{attribute 'GeneratedUsingTerminal: EL3041-0000-0017'}
{attribute addProperty BoxType "EL3041-0000-0017"}
{attribute addProperty Id "AI_StandardAT %I*AI_Standard_Channel_4A3944819WcStateAT %I*WcState_9091E0EB2InfoDataAT %I*InfoData_94A18F5E2"}
{attribute addProperty CRC "1943597556"}
{attribute addProperty Size "13"}
TYPE EL3041_73D8F1F4 EXTENDS EtcSlaveTerminalBase_947E5A46 :
STRUCT
	{attribute addProperty Name "AI_Standard"}
	AI_Standard : AI_Standard_Channel_4A394481;
	{attribute addProperty Name "WcState"}
	WcState : WcState_9091E0EB;
	{attribute addProperty Name "InfoData"}
	InfoData : InfoData_94A18F5E;
END_STRUCT
END_TYPE

(* stored: Version 1.2.0.0, ProductVersion 3.1.4024.9
   DUT EL3041_73D8F1F4: Id {d4258146-17cd-4f14-81db-79858dc6303d} *)
